% RSLogix 500 project WORKSHEET 3.RSS, saved by version 10.00.00.00 %
PROJECT "PL06B"    % processor: Bul.1763 MicroLogix 1100 Series B %

PROGRAM FILES
  LAD 2   5 rungs

DATA FILES
  O0 OUTPUT  4 elements
  I1 INPUT  6 elements
  S2 STATUS  66 elements
  B3 BINARY  1 elements
  T4 TIMER  10 elements
  C5 COUNTER  2 elements
  R6 CONTROL  1 elements
  N7 INTEGER  5 elements
  F8 FLOAT  1 elements

LADDER 2
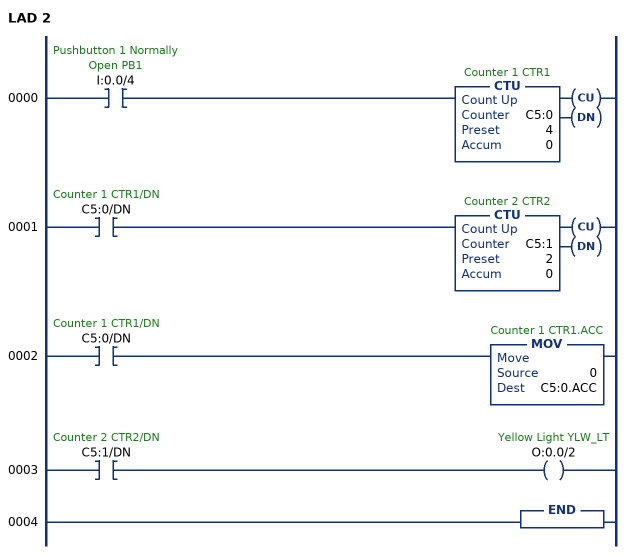
% Rung: 0 %
SOR XIC I:0.0/4 CTU C5:0 4 0 EOR
%   I:0.0/4  PB1  "Pushbutton 1 Normally Open" %
%   C5:0  CTR1  "Counter 1" %
% Rung: 1 %
SOR XIC C5:0/DN CTU C5:1 2 0 EOR
%   C5:0  CTR1  "Counter 1" %
%   C5:1  CTR2  "Counter 2" %
% Rung: 2 %
SOR XIC C5:0/DN MOV 0 C5:0.ACC EOR
%   C5:0  CTR1  "Counter 1" %
% Rung: 3 %
SOR XIC C5:1/DN OTE O:0.0/2 EOR
%   C5:1  CTR2  "Counter 2" %
%   O:0.0/2  YLW_LT  "Yellow Light" %
% Rung: 4 %
SOR END EOR

OTHER DOCUMENTED ADDRESSES
  B3:0/0  RED_ORG  "Binary Bit"
  B3:0/1  DRK_PPL  "Binary Bit"
  B3:0/2  RO_RESET  "Binary Bit"
  B3:0/3  DPL_RESET  "Binary Bit"
  B3:0/4  GRN_STOP  "Green Light 1 Stop"
  B3:0/15  SCRATCH  "Scratch Bit"
  B3:1/1  RED_TMR_DNS  "Red Light Timer Done Storage"
  I  
  I:0.0/0  SS1A  "Selector Switch 1 Position A"
  I:0.0/1  SS1B  "Selector Switch 1 Position B"
  I:0.0/2  SS2A  "Selector Switch 2 Position A"
  I:0.0/3  SS2B  "Selector Switch 2 Position B"
  I:0.0/5  PB2  "Pushbutton 2 Normally Closed"
  O:0.0/0  GRN_LT1  "Green Light 1"
  O:0.0/1  RED_LT  "Red Light"
  O:0.0/3  GRN_LT2  "Green Light 2"
  RTC:0.YR  RTC
  SEL1B  
  T4:0  RED_TMR  "Red Timer"
  T4:1  YLW_TMR  "Yellow Timer"
  T4:2  BLU_TMR  "Blue Timer"
  T4:3  RST_TMR  "Reset Timer"

DATA TABLE (non-zero values as saved)
DATA B3
% B3:0 % 0X8009
DATA T4
% .PRE .ACC %
% T4:0 % 10 0
% T4:1 % 5 0
% T4:2 % 15 0
% T4:3 % 10 0
DATA C5
% .PRE .ACC %
% C5:0 % 4 0
% C5:1 % 2 0
DATA N7
% N7:0 % 555 0 0 0 0
